(* IEC 61131-3 sources: PLC-Extruder-project/plc, 7 files *)

(* ---- ExtruderController.st ---- *)
(*
    Vendor-neutral IEC 61131-3 Structured Text translation of the
    Python ExtruderController state machine.

    Source model:
    - plc_extruder/controller.py

    Notes:
    - This block focuses on orchestration, not detailed process physics.
    - Heater, feeder, motor, die, and safety logic are expected to live
      in separate PLC function blocks.
    - Commands such as StartCmd/StopCmd/ResetCmd are edge-triggered.
    - Maintained outputs are derived from State each scan.
*)

TYPE E_ControllerState :
(
    IDLE,
    STARTUP,
    RUNNING,
    SHUTDOWN,
    EMERGENCY_STOP
);
END_TYPE

FUNCTION_BLOCK FB_ExtruderController
VAR_INPUT
    StartCmd : BOOL;
    StopCmd : BOOL;
    ResetCmd : BOOL;
    EmergencyStopCmd : BOOL;

    SafetyEStop : BOOL;
    HeaterAllAtSetpoint : BOOL;
    DieAtSetpoint : BOOL;
    MotorActualRpm : REAL;

    RecipeFeedRateCmd : REAL := 50.0;
    RecipeScrewRpmCmd : REAL := 80.0;
    FeedRateMin : REAL := 5.0;
    FeedRateMax : REAL := 100.0;
    ScrewRpmMin : REAL := 5.0;
    ScrewRpmMax : REAL := 150.0;

    CycleTime_s : REAL := 0.1;
END_VAR
VAR_OUTPUT
    State : E_ControllerState := IDLE;
    ScanNumber : DINT := 0;
    RunTime_s : REAL := 0.0;

    FeedRateSetpoint : REAL := 5.0;
    ScrewRpmSetpoint : REAL := 5.0;

    HeaterEnableCmd : BOOL := FALSE;
    DieEnableCmd : BOOL := FALSE;
    FeederRunCmd : BOOL := FALSE;
    MotorRunCmd : BOOL := FALSE;

    ResetSafetyCmd : BOOL := FALSE;
    ResetMotorFaultCmd : BOOL := FALSE;
    ResetFeederFaultCmd : BOOL := FALSE;

    RaiseShutdownAlarmCmd : BOOL := FALSE;
    ClearShutdownAlarmCmd : BOOL := FALSE;
    RaiseEStopAlarmCmd : BOOL := FALSE;
END_VAR
VAR
    PrevState : E_ControllerState := IDLE;

    StartCmdPrev : BOOL := FALSE;
    StopCmdPrev : BOOL := FALSE;
    ResetCmdPrev : BOOL := FALSE;
    EmergencyStopCmdPrev : BOOL := FALSE;

    StartEdge : BOOL := FALSE;
    StopEdge : BOOL := FALSE;
    ResetEdge : BOOL := FALSE;
    EmergencyStopEdge : BOOL := FALSE;
END_VAR

(* Reset one-scan pulse outputs *)
ResetSafetyCmd := FALSE;
ResetMotorFaultCmd := FALSE;
ResetFeederFaultCmd := FALSE;
RaiseShutdownAlarmCmd := FALSE;
ClearShutdownAlarmCmd := FALSE;
RaiseEStopAlarmCmd := FALSE;

(* Rising-edge detection *)
StartEdge := StartCmd AND NOT StartCmdPrev;
StopEdge := StopCmd AND NOT StopCmdPrev;
ResetEdge := ResetCmd AND NOT ResetCmdPrev;
EmergencyStopEdge := EmergencyStopCmd AND NOT EmergencyStopCmdPrev;

StartCmdPrev := StartCmd;
StopCmdPrev := StopCmd;
ResetCmdPrev := ResetCmd;
EmergencyStopCmdPrev := EmergencyStopCmd;

(* Scan bookkeeping *)
ScanNumber := ScanNumber + 1;

(* Recipe clamping *)
FeedRateSetpoint := MAX(FeedRateMin, MIN(RecipeFeedRateCmd, FeedRateMax));
ScrewRpmSetpoint := MAX(ScrewRpmMin, MIN(RecipeScrewRpmCmd, ScrewRpmMax));

(* High-priority safety transition *)
IF ((SafetyEStop OR EmergencyStopEdge) AND (State <> EMERGENCY_STOP) AND (State <> IDLE)) THEN
    State := EMERGENCY_STOP;
END_IF;

(* Operator transitions *)
CASE State OF
    IDLE:
        IF StartEdge THEN
            RunTime_s := 0.0;
            State := STARTUP;
        ELSIF ResetEdge THEN
            RunTime_s := 0.0;
            ResetSafetyCmd := TRUE;
            ResetMotorFaultCmd := TRUE;
            ResetFeederFaultCmd := TRUE;
        END_IF;

    STARTUP:
        IF StopEdge THEN
            State := SHUTDOWN;
        ELSIF HeaterAllAtSetpoint AND DieAtSetpoint THEN
            State := RUNNING;
        END_IF;

    RUNNING:
        IF StopEdge THEN
            State := SHUTDOWN;
        ELSIF SafetyEStop OR EmergencyStopEdge THEN
            State := EMERGENCY_STOP;
        ELSE
            RunTime_s := RunTime_s + CycleTime_s;
        END_IF;

    SHUTDOWN:
        IF SafetyEStop OR EmergencyStopEdge THEN
            State := EMERGENCY_STOP;
        ELSIF MotorActualRpm < 0.5 THEN
            State := IDLE;
            ClearShutdownAlarmCmd := TRUE;
        END_IF;

    EMERGENCY_STOP:
        IF ResetEdge THEN
            RunTime_s := 0.0;
            ResetSafetyCmd := TRUE;
            ResetMotorFaultCmd := TRUE;
            ResetFeederFaultCmd := TRUE;
            ClearShutdownAlarmCmd := TRUE;
            State := IDLE;
        END_IF;
END_CASE;

(* State entry actions *)
IF State <> PrevState THEN
    CASE State OF
        STARTUP:
            RunTime_s := 0.0;

        RUNNING:
            (* Recipe setpoints are already exposed as maintained outputs. *)

        SHUTDOWN:
            RaiseShutdownAlarmCmd := TRUE;

        EMERGENCY_STOP:
            RaiseEStopAlarmCmd := TRUE;

        IDLE:
            (* Outputs are handled below as maintained state outputs. *)
    END_CASE;

    PrevState := State;
END_IF;

(* Maintained outputs by state *)
HeaterEnableCmd := (State = STARTUP) OR (State = RUNNING) OR (State = SHUTDOWN);
DieEnableCmd := (State = STARTUP) OR (State = RUNNING) OR (State = SHUTDOWN);
FeederRunCmd := (State = RUNNING);
MotorRunCmd := (State = RUNNING);

END_FUNCTION_BLOCK

(* ---- FB_DieZone.st ---- *)
(*
    Generic die-zone function block for IEC 61131-3 Structured Text.

    Handles:
    - die temperature command
    - melt pressure estimation
    - throughput estimation
    - over-temperature and over-pressure alarms
*)

FUNCTION_BLOCK FB_DieZone
VAR_INPUT
    EnableCmd : BOOL;
    ResetCmd : BOOL;
    TemperaturePV : REAL;
    Setpoint : REAL := 235.0;
    TempTolerance : REAL := 5.0;
    MaxTemp : REAL := 280.0;

    ScrewRpmPV : REAL;
    FeedRateActualKgH : REAL;
    MotorMaxRpm : REAL := 150.0;
    DieOpeningPct : REAL := 100.0;
    PressureCoef : REAL := 1.8;
    DieMaxPressureBar : REAL := 350.0;
    DieWarningPressureBar : REAL := 300.0;

    Kp : REAL := 3.0;
END_VAR
VAR_OUTPUT
    HeaterEnable : BOOL := FALSE;
    HeaterOutputPct : REAL := 0.0;
    AtSetpoint : BOOL := FALSE;
    MeltPressureBar : REAL := 0.0;
    ThroughputKgH : REAL := 0.0;
    OverTempAlarm : BOOL := FALSE;
    OverPressureAlarm : BOOL := FALSE;
    HighPressureWarning : BOOL := FALSE;
END_VAR
VAR
    TempError : REAL := 0.0;
    EffectiveOpeningPct : REAL := 100.0;
    ViscosityFactor : REAL := 1.0;
END_VAR

IF ResetCmd THEN
    OverTempAlarm := FALSE;
    OverPressureAlarm := FALSE;
    HighPressureWarning := FALSE;
END_IF;

HeaterEnable := EnableCmd;
AtSetpoint := ABS(TemperaturePV - Setpoint) <= TempTolerance;

IF NOT EnableCmd THEN
    HeaterOutputPct := 0.0;
ELSE
    IF TemperaturePV >= MaxTemp THEN
        OverTempAlarm := TRUE;
        HeaterOutputPct := 0.0;
    ELSE
        TempError := Setpoint - TemperaturePV;
        HeaterOutputPct := LIMIT(0.0, TempError * Kp, 100.0);
    END_IF;
END_IF;

EffectiveOpeningPct := LIMIT(5.0, DieOpeningPct, 100.0);

IF ScrewRpmPV <= 0.0 THEN
    MeltPressureBar := 0.0;
    ThroughputKgH := 0.0;
ELSE
    ViscosityFactor := LIMIT(0.2, 1.0 - ((TemperaturePV - 100.0) / 300.0), 1.0);
    MeltPressureBar := PressureCoef * ScrewRpmPV * ViscosityFactor / (EffectiveOpeningPct / 100.0);
    MeltPressureBar := LIMIT(0.0, MeltPressureBar, DieMaxPressureBar * 1.1);

    IF MotorMaxRpm > 0.0 THEN
        ThroughputKgH := FeedRateActualKgH * (ScrewRpmPV / MotorMaxRpm);
    ELSE
        ThroughputKgH := 0.0;
    END_IF;
END_IF;

OverPressureAlarm := MeltPressureBar >= DieMaxPressureBar;
HighPressureWarning := MeltPressureBar >= DieWarningPressureBar;

END_FUNCTION_BLOCK

(* ---- FB_ExtrusionMotor.st ---- *)
(*
    Generic extrusion-motor/VFD function block for IEC 61131-3 Structured Text.

    Handles:
    - speed reference command
    - estimated load / current supervision
    - overspeed and overcurrent interlocks
*)

FUNCTION_BLOCK FB_ExtrusionMotor
VAR_INPUT
    RunCmd : BOOL;
    ResetCmd : BOOL;
    SpeedSetpointRpm : REAL := 80.0;
    ActualRpmPV : REAL;
    MeltPressureBar : REAL;
    MinRpm : REAL := 5.0;
    MaxRpm : REAL := 150.0;
    RatedCurrentA : REAL := 100.0;
    CurrentLimitA : REAL := 100.0;
    MaxTorquePct : REAL := 120.0;
    DieMaxPressureBar : REAL := 350.0;
    BackpressureCoef : REAL := 0.6;
    Kp : REAL := 1.5;
END_VAR
VAR_OUTPUT
    MotorEnable : BOOL := FALSE;
    SpeedCommandRpm : REAL := 5.0;
    VfdOutputPct : REAL := 0.0;
    TorquePct : REAL := 0.0;
    CurrentEstimateA : REAL := 0.0;
    OverCurrentAlarm : BOOL := FALSE;
    OverSpeedAlarm : BOOL := FALSE;
    StallWarning : BOOL := FALSE;
    FaultActive : BOOL := FALSE;
END_VAR
VAR
    SpeedError : REAL := 0.0;
    SpeedLoadPct : REAL := 0.0;
    PressureLoadPct : REAL := 0.0;
END_VAR

IF ResetCmd THEN
    OverCurrentAlarm := FALSE;
    OverSpeedAlarm := FALSE;
    StallWarning := FALSE;
    FaultActive := FALSE;
END_IF;

SpeedCommandRpm := LIMIT(MinRpm, SpeedSetpointRpm, MaxRpm);

IF RunCmd AND NOT FaultActive THEN
    MotorEnable := TRUE;
    SpeedError := SpeedCommandRpm - ActualRpmPV;
    VfdOutputPct := LIMIT(0.0, SpeedError * Kp, 100.0);
ELSE
    MotorEnable := FALSE;
    VfdOutputPct := 0.0;
END_IF;

IF MaxRpm > 0.0 THEN
    SpeedLoadPct := (ActualRpmPV / MaxRpm) * 40.0;
ELSE
    SpeedLoadPct := 0.0;
END_IF;

IF DieMaxPressureBar > 0.0 THEN
    PressureLoadPct := (MeltPressureBar / DieMaxPressureBar) * 60.0;
ELSE
    PressureLoadPct := 0.0;
END_IF;

TorquePct := LIMIT(0.0, SpeedLoadPct + (PressureLoadPct * BackpressureCoef), 100.0);
CurrentEstimateA := (TorquePct / 100.0) * RatedCurrentA;

OverCurrentAlarm := CurrentEstimateA >= CurrentLimitA;
OverSpeedAlarm := ActualRpmPV > (MaxRpm * 1.05);
StallWarning := TorquePct >= MaxTorquePct;

IF OverCurrentAlarm OR OverSpeedAlarm THEN
    FaultActive := TRUE;
END_IF;

END_FUNCTION_BLOCK

(* ---- FB_HeatingZone.st ---- *)
(*
    Generic heating-zone function block for IEC 61131-3 Structured Text.

    Intended use:
    - One instance per barrel zone
    - Real PLC input should be the measured process temperature
    - Real PLC output should drive heater SSR/contactors and cooling valve/fan

    Note:
    - This uses a simple proportional control law as a portable baseline.
    - Replace the proportional section with your platform's PID block if needed.
*)

FUNCTION_BLOCK FB_HeatingZone
VAR_INPUT
    EnableCmd : BOOL;
    ResetCmd : BOOL;
    TemperaturePV : REAL;
    Setpoint : REAL := 200.0;
    TempTolerance : REAL := 5.0;
    MaxTemp : REAL := 280.0;
    UnderTempBand : REAL := 20.0;
    Kp : REAL := 3.0;
END_VAR
VAR_OUTPUT
    HeaterEnable : BOOL := FALSE;
    HeaterOutputPct : REAL := 0.0;
    CoolingOutputPct : REAL := 0.0;
    AtSetpoint : BOOL := FALSE;
    OverTempAlarm : BOOL := FALSE;
    UnderTempAlarm : BOOL := FALSE;
END_VAR
VAR
    TempError : REAL := 0.0;
END_VAR

IF ResetCmd THEN
    OverTempAlarm := FALSE;
    UnderTempAlarm := FALSE;
END_IF;

HeaterEnable := EnableCmd;
AtSetpoint := ABS(TemperaturePV - Setpoint) <= TempTolerance;

IF NOT EnableCmd THEN
    HeaterOutputPct := 0.0;
    CoolingOutputPct := 0.0;
ELSIF TemperaturePV >= MaxTemp THEN
    OverTempAlarm := TRUE;
    HeaterOutputPct := 0.0;
    CoolingOutputPct := 100.0;
ELSE
    TempError := Setpoint - TemperaturePV;
    HeaterOutputPct := LIMIT(0.0, TempError * Kp, 100.0);

    IF TempError < (-1.0 * TempTolerance) THEN
        CoolingOutputPct := LIMIT(0.0, ABS(TempError) * 5.0, 100.0);
    ELSE
        CoolingOutputPct := 0.0;
    END_IF;

    IF TemperaturePV < (Setpoint - UnderTempBand) THEN
        UnderTempAlarm := TRUE;
    ELSE
        UnderTempAlarm := FALSE;
    END_IF;
END_IF;

END_FUNCTION_BLOCK

(* ---- FB_MaterialFeeder.st ---- *)
(*
    Generic material-feeder function block for IEC 61131-3 Structured Text.

    Handles:
    - run command and drive reference
    - hopper level alarms
    - empty-hopper fault interlock
*)

FUNCTION_BLOCK FB_MaterialFeeder
VAR_INPUT
    RunCmd : BOOL;
    ResetCmd : BOOL;
    FeedRateSetpointKgH : REAL := 50.0;
    ActualRatePVKgH : REAL;
    HopperLevelPctPV : REAL := 100.0;
    MinRateKgH : REAL := 5.0;
    MaxRateKgH : REAL := 100.0;
    LowLevelPct : REAL := 10.0;
    EmptyLevelPct : REAL := 2.0;
    Kp : REAL := 2.0;
END_VAR
VAR_OUTPUT
    FeederEnable : BOOL := FALSE;
    DriveOutputPct : REAL := 0.0;
    FeedRateCommandKgH : REAL := 5.0;
    LowMaterialAlarm : BOOL := FALSE;
    EmptyHopperAlarm : BOOL := FALSE;
    FaultActive : BOOL := FALSE;
END_VAR
VAR
    RateError : REAL := 0.0;
END_VAR

IF ResetCmd THEN
    EmptyHopperAlarm := FALSE;
    FaultActive := FALSE;
END_IF;

FeedRateCommandKgH := LIMIT(MinRateKgH, FeedRateSetpointKgH, MaxRateKgH);
LowMaterialAlarm := HopperLevelPctPV <= LowLevelPct;

IF HopperLevelPctPV <= EmptyLevelPct THEN
    EmptyHopperAlarm := TRUE;
    FaultActive := TRUE;
END_IF;

IF RunCmd AND NOT FaultActive THEN
    FeederEnable := TRUE;
    RateError := FeedRateCommandKgH - ActualRatePVKgH;
    DriveOutputPct := LIMIT(0.0, RateError * Kp, 100.0);
ELSE
    FeederEnable := FALSE;
    DriveOutputPct := 0.0;
END_IF;

END_FUNCTION_BLOCK

(* ---- FB_SafetySystem.st ---- *)
(*
    Generic safety/interlock function block for IEC 61131-3 Structured Text.

    This block consolidates:
    - hardware and software E-stop
    - temperature / pressure / drive-fault interlocks
    - watchdog supervision input from a higher-level task
*)

TYPE E_SafetyState :
(
    SAFE,
    WARNING,
    E_STOP
);
END_TYPE

FUNCTION_BLOCK FB_SafetySystem
VAR_INPUT
    ResetCmd : BOOL;
    HardwareEStop : BOOL;
    SoftwareEStop : BOOL;
    AnyZoneOverTemp : BOOL;
    DieOverPressure : BOOL;
    MotorFault : BOOL;
    WarningPresent : BOOL;
    WatchdogHealthy : BOOL := TRUE;
END_VAR
VAR_OUTPUT
    State : E_SafetyState := SAFE;
    EStopActive : BOOL := FALSE;
    InterlockTempAlarm : BOOL := FALSE;
    InterlockPressureAlarm : BOOL := FALSE;
    InterlockMotorAlarm : BOOL := FALSE;
    WatchdogAlarm : BOOL := FALSE;
END_VAR

IF ResetCmd THEN
    InterlockTempAlarm := FALSE;
    InterlockPressureAlarm := FALSE;
    InterlockMotorAlarm := FALSE;
    WatchdogAlarm := FALSE;
    EStopActive := FALSE;
    State := SAFE;
END_IF;

IF AnyZoneOverTemp THEN
    InterlockTempAlarm := TRUE;
END_IF;

IF DieOverPressure THEN
    InterlockPressureAlarm := TRUE;
END_IF;

IF MotorFault THEN
    InterlockMotorAlarm := TRUE;
END_IF;

IF NOT WatchdogHealthy THEN
    WatchdogAlarm := TRUE;
END_IF;

EStopActive :=
    HardwareEStop OR
    SoftwareEStop OR
    InterlockTempAlarm OR
    InterlockPressureAlarm OR
    InterlockMotorAlarm OR
    WatchdogAlarm;

IF EStopActive THEN
    State := E_STOP;
ELSIF WarningPresent THEN
    State := WARNING;
ELSE
    State := SAFE;
END_IF;

END_FUNCTION_BLOCK

(* ---- ExtruderCellExample.st ---- *)
(*
    Example top-level program wiring the PLC function blocks together.

    This is a guide for integration, not a finished hardware project.
    Replace TempPV/RpmPV/LevelPV variables with real I/O or mapped tags.
*)

PROGRAM PRG_ExtruderCell
VAR
    Ctrl : FB_ExtruderController;
    Zone1 : FB_HeatingZone;
    Zone2 : FB_HeatingZone;
    Zone3 : FB_HeatingZone;
    Zone4 : FB_HeatingZone;
    Die : FB_DieZone;
    Feeder : FB_MaterialFeeder;
    Motor : FB_ExtrusionMotor;
    Safety : FB_SafetySystem;

    StartPB : BOOL;
    StopPB : BOOL;
    ResetPB : BOOL;
    EStopPB : BOOL;

    Z1TempPV : REAL;
    Z2TempPV : REAL;
    Z3TempPV : REAL;
    Z4TempPV : REAL;
    DieTempPV : REAL;
    MotorRpmPV : REAL;
    FeederRatePV : REAL;
    HopperLevelPctPV : REAL;
END_VAR

Zone1(
    EnableCmd := Ctrl.HeaterEnableCmd,
    ResetCmd := Ctrl.ResetSafetyCmd,
    TemperaturePV := Z1TempPV,
    Setpoint := 180.0
);
Zone2(
    EnableCmd := Ctrl.HeaterEnableCmd,
    ResetCmd := Ctrl.ResetSafetyCmd,
    TemperaturePV := Z2TempPV,
    Setpoint := 200.0
);
Zone3(
    EnableCmd := Ctrl.HeaterEnableCmd,
    ResetCmd := Ctrl.ResetSafetyCmd,
    TemperaturePV := Z3TempPV,
    Setpoint := 220.0
);
Zone4(
    EnableCmd := Ctrl.HeaterEnableCmd,
    ResetCmd := Ctrl.ResetSafetyCmd,
    TemperaturePV := Z4TempPV,
    Setpoint := 230.0
);

Feeder(
    RunCmd := Ctrl.FeederRunCmd,
    ResetCmd := Ctrl.ResetFeederFaultCmd,
    FeedRateSetpointKgH := Ctrl.FeedRateSetpoint,
    ActualRatePVKgH := FeederRatePV,
    HopperLevelPctPV := HopperLevelPctPV
);

Die(
    EnableCmd := Ctrl.DieEnableCmd,
    ResetCmd := Ctrl.ResetSafetyCmd,
    TemperaturePV := DieTempPV,
    ScrewRpmPV := MotorRpmPV,
    FeedRateActualKgH := FeederRatePV
);

Motor(
    RunCmd := Ctrl.MotorRunCmd,
    ResetCmd := Ctrl.ResetMotorFaultCmd,
    SpeedSetpointRpm := Ctrl.ScrewRpmSetpoint,
    ActualRpmPV := MotorRpmPV,
    MeltPressureBar := Die.MeltPressureBar
);

Safety(
    ResetCmd := Ctrl.ResetSafetyCmd,
    HardwareEStop := EStopPB,
    SoftwareEStop := FALSE,
    AnyZoneOverTemp :=
        Zone1.OverTempAlarm OR
        Zone2.OverTempAlarm OR
        Zone3.OverTempAlarm OR
        Zone4.OverTempAlarm,
    DieOverPressure := Die.OverPressureAlarm,
    MotorFault := Motor.FaultActive,
    WarningPresent :=
        Zone1.UnderTempAlarm OR
        Zone2.UnderTempAlarm OR
        Zone3.UnderTempAlarm OR
        Zone4.UnderTempAlarm OR
        Die.HighPressureWarning OR
        Feeder.LowMaterialAlarm OR
        Motor.StallWarning,
    WatchdogHealthy := TRUE
);

Ctrl(
    StartCmd := StartPB,
    StopCmd := StopPB,
    ResetCmd := ResetPB,
    EmergencyStopCmd := FALSE,
    SafetyEStop := Safety.EStopActive,
    HeaterAllAtSetpoint :=
        Zone1.AtSetpoint AND
        Zone2.AtSetpoint AND
        Zone3.AtSetpoint AND
        Zone4.AtSetpoint,
    DieAtSetpoint := Die.AtSetpoint,
    MotorActualRpm := MotorRpmPV,
    RecipeFeedRateCmd := 50.0,
    RecipeScrewRpmCmd := 80.0,
    CycleTime_s := 0.1
);

END_PROGRAM
